(* IEC 61131-3 sources: CannyIEC/extracted_st, 10 files *)

(* ---- ERROR.st ---- *)
(* --- Interface --- *)
{attribute 'qualified_only'}
//{attribute 'conditionalshow'}
//{attribute 'conditionalshow' := 'SomeText'}
//{attribute 'hide'}
TYPE ERROR : (
        NO_ERROR,
        TIME_OUT
    );
END_TYPE

(* ---- Constants.st ---- *)
(* --- Interface --- *)
{attribute 'qualified_only'}
//{attribute 'conditionalshow'}
//{attribute 'conditionalshow' := 'SomeText'}
//{attribute 'hide'}
VAR_GLOBAL CONSTANT
    gc_iDummy : INT := 42; /// This is a dummy global constant variable
END_VAR

(* ---- Variables.st ---- *)
(* --- Interface --- *)

{attribute 'qualified_only'}
//{attribute 'conditionalshow'}
//{attribute 'conditionalshow' := 'SomeText'}
//{attribute 'hide'}
VAR_GLOBAL
    g_iDummy : INT; /// This is a dummy global variable
END_VAR

(* ---- GetLibVersion.st ---- *)
(* --- Interface --- *)
// This function has been automatically generated from the project information.
FUNCTION GetLibVersion : VERSION
VAR_INPUT

END_VAR
(* --- Implementation --- *)
GetLibVersion.uiMajor := 0;
GetLibVersion.uiMinor := 1;
GetLibVersion.uiServicePack := 11;
GetLibVersion.uiPatch := 10;

(* ---- GetLibVersionNumber.st ---- *)
(* --- Interface --- *)
// This function has been automatically generated from the project information.
FUNCTION GetLibVersionNumber : DWORD
VAR_INPUT

END_VAR
(* --- Implementation --- *)
GetLibVersionNumber := 68362;

(* ---- ISIGNBIT.st ---- *)
(* --- Interface --- *)

FUNCTION ISIGNBIT : BIT
VAR_INPUT
    iValue : INT;
END_VAR

(* --- Implementation --- *)

ISIGNBIT := iValue < INT#0;

(* ---- IsLibReleased.st ---- *)
(* --- Interface --- *)
// This function has been automatically generated from the project information.
FUNCTION IsLibReleased : BOOL
VAR_INPUT

END_VAR
(* --- Implementation --- *)
IsLibReleased := FALSE;

(* ---- REPSILONEQ.st ---- *)
(* --- Interface --- *)
FUNCTION REPSILONEQ : BOOL
VAR_INPUT
    rLHS     : REAL;
    rRHS     : REAL;
    rEpsilon : REAL;
END_VAR

(* --- Implementation --- *)
(* Should real-epsilon comparison use "less than, or "less than or equal
to"? What should happen on the epsilon boundary? At its extreme, epsilon
is the smallest possible difference representable in the system.

In addition, what happens if rEpsilon is zero, or even negative? *)
REPSILONEQ := ABS(rLHS - rRHS) < rEpsilon;

(* ---- RSIGNBIT.st ---- *)
(* --- Interface --- *)

FUNCTION RSIGNBIT : BIT
VAR_INPUT
    rValue : REAL;
END_VAR

(* --- Implementation --- *)

RSIGNBIT := rValue < REAL#0;

(* ---- SymmetricDebounce.st ---- *)
(* --- Interface --- *)

FUNCTION_BLOCK SymmetricDebounce
VAR_INPUT
    xDirty: BOOL; (* raw input signal from a sensor or switch *)
END_VAR
VAR_OUTPUT
    xClean: BOOL; (* debounced "input" signal *)
END_VAR
VAR
    tPresetFalling: TIME; (* preset time for falling edge debounce *)
    tPresetRising: TIME; (* preset time for rising edge debounce *)
    tPreset: TIME := T#50ms; (* symmetric preset time used if specific rising/falling presets are not set; default to 50 milliseconds *)
    fbDelayedRising: TON; (* timer for rising edge *)
    fbDelayedFalling: TOF; (* timer for falling edge *)
END_VAR

(* --- Implementation --- *)

(* The raw input signal passes through the TON and TOF function blocks, which
implement the debounce logic. The TON block starts timing when the raw input
goes high, and the TOF block starts timing when the TON output goes low. The
system takes the debounced output signal from the TOF output. *)
(* Rising edge debounce *)
fbDelayedRising(IN := xDirty, PT := SEL(tPresetRising <> T#0s, tPresetRising, tPreset));
(* Falling edge debounce *)
fbDelayedFalling(IN := fbDelayedRising.Q, PT := SEL(tPresetFalling <> T#0s, tPresetFalling, tPreset));
xClean := fbDelayedFalling.Q;
